FUNCTION F_CheckIndexBounds_UINT : UINT
VAR_INPUT
	lowerbound		: 	UINT;
	upperbound		:   UINT;
END_VAR
VAR_IN_OUT
	index			: 	UINT;
END_VAR

IF  index < lowerbound THEN
	F_CheckIndexBounds_UINT := lowerbound;
	index 		:= lowerbound;
ELSIF  index > upperbound THEN
	F_CheckIndexBounds_UINT := upperbound;
	index 		:= upperbound;
ELSE  
	F_CheckIndexBounds_UINT := index;
END_IF

END_FUNCTION

(* stored: Version 1.1.0.1, ProductVersion 3.1.4024.3
   POU F_CheckIndexBounds_UINT: Id {96149f12-593a-4afb-afbd-0fdc972bcc75}, SpecialFunc None *)
